{attribute addProperty BoxType "EL2024-0000-0016"}
{attribute addProperty Id "ChannelAT %Q*ARRAY[0..3] OF Channel_7F374EB03240WcStateAT %I*WcState_64F6A8C6810InfoDataAT %I*InfoData_192954DE1620"}
{attribute addProperty CRC "999552494"}
{attribute addProperty SizeInBites "56"}
{attribute addProperty SizeInBytes "7"}
TYPE EL2024_E7E37CC2 :
STRUCT
	{attribute addProperty Name "Channel"}
	Channel : ARRAY[0..3] OF Channel_7F374EB0;
	{attribute addProperty Name "WcState"}
	WcState : WcState_64F6A8C6;
	{attribute addProperty Name "InfoData"}
	InfoData : InfoData_192954DE;
END_STRUCT
END_TYPE

(* stored: Version 1.2.0.0, ProductVersion 3.1.4024.9
   DUT EL2024_E7E37CC2: Id {19eaaed0-3a79-407a-85ca-f9d8f4aaacc4} *)
